// TIA Portal V17 export
// export: Created 2025-03-05T08:01:00.5358223Z, ExportSetting WithDefaults, DisplayName Totally Integrated Automation Portal, DisplayVersion V17 Update 8, DisplayName TIA Portal Openness, DisplayVersion V17 Update 8, DisplayName TIA Portal Version Control Interface, DisplayVersion V17, DisplayName SINAMICS Startdrive Advanced, DisplayVersion V17 SP2, DisplayName SINAMICS Startdrive G110M, G120, G120C, G120D, G120P, G115D, DisplayVersion V17 SP2, DisplayName SINAMICS Startdrive G130, G150, S120, S150, SINAMICS MV, S210, DisplayVersion V17 SP2, DisplayName STEP 7 Professional, DisplayVersion V17 Update 8, DisplayName SINUMERIK ONE STEP 7 Toolbox, DisplayVersion V17 Update 12, DisplayName SINUMERIK 840D sl STEP 7 Toolbox, DisplayVersion V17 Update 12, DisplayName STEP 7 Safety, DisplayVersion V17 Update 6, DisplayName WinCC Advanced, DisplayVersion V17 Update 8
DATA_BLOCK "LTLP_DeviceInterfaceData"   // DB546
{ S7_Optimized_Access := 'FALSE'; DB_Accessible_From_OPC_UA := 'FALSE' }
VERSION : 0.1
// stored: AutoNumber true, DBAccessibleFromOPCUA false, DBAccessibleFromWebserver true, InstanceOfName LTLP_typeDeviceInterface, InstanceOfType UDT, IsOnlyStoredInLoadMemory false, IsWriteProtectedInAS false
"LTLP_typeDeviceInterface"
   // VAR RETAIN
   //    inputs : Struct
   //       mppFunctions { S7_SetPoint := 'True'} : "LTLP_typeMppFunctions";
   //       mcpFunctions { S7_SetPoint := 'True'} : "LTLP_typeMcpFunctions";
   //       mcpFctAdd : Struct
   //          feed_correction : Byte;
   //          spindle_correction : Byte;
   //          protection_level : Byte;
   //          authorization : Byte;
   //       END_STRUCT;
   //       axes : Array[1..31] of Bool;
   //       oemFunctions : Array[1..100] of Bool;
   //    END_STRUCT;
   //    outputs : Struct
   //       mppFunctions { S7_SetPoint := 'True'} : "LTLP_typeMppFunctions";
   //       mcpFunctions { S7_SetPoint := 'True'} : "LTLP_typeMcpFunctions";
   //       mcpFctAdd : Struct
   //          feed_correction : Byte;
   //          spindle_correction : Byte;
   //          protection_level : Byte;
   //          authorization : Byte;
   //       END_STRUCT;
   //       axisNo : Array[1..31] of Bool;
   //       axisIsGeoAxis : Bool;
   //       oemFunctions : Array[1..100] of Bool;
   //    END_STRUCT;
   //    edgeNegEnableMpp : Bool;
   //    edgeNegKeyLocked : Bool;
   //    mppConnected : Bool;
   //    mcpConnected : Bool;
   //    ht8Connected : Bool;
   //    ht2Connected : Bool;
   //    mppDAGConnected : Bool;
   //    ht2Active : Bool;
   //    keyPressed : Bool;
   //    internalStorageData : Struct
   //       negTriggerLampTestMpp : Bool;
   //       negTriggerLampTestMcp : Bool;
   //       negTriggerLampTestHt8 : Bool;
   //       negTriggerLampTestHt2 : Bool;
   //       negTriggerLampTestAxisSel : Bool;
   //       posTriggerTimeTckRead : Bool;
   //       actualTimeTckSaved : Time;
   //    END_STRUCT;
   // END_VAR
BEGIN
END_DATA_BLOCK
